# B&R Automation Studio project AS_Target_Simulink_Test (part 2)

### sfc_sdi.h
```c
/* Copyright 2013-2014 The MathWorks, Inc. */

#ifndef _sf_runtime_sf_sdi_h_
#define _sf_runtime_sf_sdi_h_

#ifdef SUPPORTS_PRAGMA_ONCE
#pragma once
#endif

#include "sf_runtime_spec.h"

typedef enum {
    SF_DATA_MODE = 0,
    SF_CHILD_ACTIVITY_MODE  = 0x01,
    SF_LEAF_ACTIVITY_MODE   = 0x02,
    SF_SELF_ACTIVITY_MODE   = 0x04
} SFSdiModeFlag;

typedef enum {
    SF_DATA_TYPE_BEGIN = 0,
    SF_DATA_TYPE_DOUBLE = SF_DATA_TYPE_BEGIN,
    SF_DATA_TYPE_SINGLE,
    SF_DATA_TYPE_INT8,
    SF_DATA_TYPE_UINT8,
    SF_DATA_TYPE_INT16,
    SF_DATA_TYPE_UINT16,
    SF_DATA_TYPE_INT32,
    SF_DATA_TYPE_UINT32,
    SF_DATA_TYPE_BOOLEAN,
    SF_DATA_TYPE_LAST
} SF2SdiBuiltInDataTypes;

typedef enum {
    SF_DIMENSIONS_BEGIN = 0,
    SF_DIMENSIONS_MODE_FIXED = SF_DIMENSIONS_BEGIN,
    SF_DIMENSIONS_MODE_VARIABLE,
    SF_DIMENSIONS_LAST
} SF2SdiDimsMode;

typedef enum {
    SF_COMPLEXITY_BEGIN = 0,
    SF_REAL = SF_COMPLEXITY_BEGIN,
    SF_COMPLEX,
    SF_COMPLEXITY_LAST
} SF2SdiComplexity;

typedef enum {
    SF_SAMPLE_TIME_BEGIN = 0,
    SF_SAMPLE_TIME_CONTINUOUS = SF_SAMPLE_TIME_BEGIN,
    SF_SAMPLE_TIME_DISCRETE,
    SF_SAMPLE_TIME_LAST
} SF2SdiUpdateMethod;

typedef struct SignalExportStruct_t {
    int useCustomName;
    int limitDataPoints;
    int decimate;
    const char* logName;
    const char* signalName;
    unsigned int maxPoints;
    unsigned int decimation;
} SignalExportStruct;

typedef struct sdiBlockID {
    void* SimStruct;
    char* mdlRefFullPath;
    char* blkPath;
    void* sdiRuntime;
} sdiBlockID_t;

LIBMWSF_RUNTIME_API void sdi_database_initialize(struct sdiBlockID* blockId,
                                                 unsigned int* stateSSIDs,
                                                 uint8_T* loggedStatesBuffer, int numStates,
                                                 unsigned int* dataSSIDs,
                                                 uint8_T* loggedDataBuffer, int numData);

LIBMWSF_RUNTIME_API void sdi_database_terminate(struct sdiBlockID* blockId);

LIBMWSF_RUNTIME_API void sdi_register_self_activity_signal(
    struct sdiBlockID* blockId,
    const char* targetName,
    const char* ssid,
    int uMethod,
    SignalExportStruct *sigExportProps,
    unsigned int ssId);

LIBMWSF_RUNTIME_API void sdi_register_child_activity_signal(
    struct sdiBlockID* blockId,
    const char* targetName,
    const char* parentStateRelativePath,
    int numChildStates,
    const char** stateNames,
    int* values,
    int signalSize,
    int uMethod,
    unsigned int ssId);

LIBMWSF_RUNTIME_API void sdi_register_leaf_activity_signal(
    struct sdiBlockID* blockId,
    const char* targetName,
    const char* parentStateRelativePath,
    int numLeafStates,
    const char** stateNames,
    int* values,
    int signalSize,
    int uMethod,
    unsigned int ssId);

LIBMWSF_RUNTIME_API void sdi_register_enum_data_type_signal(
    struct sdiBlockID* blockId,
    const char* targetName,
    const char* parentStateRelativePath,
    const char* enumTypeName,
    int numLiterals,
    const char** literals,
    int* enumValues,
    int storageSize, int isSigned,
    int numDims, int* dimsArray,
    int uMethod,
    int dimsMode,
    int complexity,
    SignalExportStruct *sigExportProps,
    unsigned int ssId);

LIBMWSF_RUNTIME_API void sdi_register_builtin_data_type_signal(
    struct sdiBlockID* blockId,
    const char* targetName,
    const char* parentStateRelativePath,
    int numDims,
    int* dims,
    int updateMethod,
    int typ,
    int dimsMode,
    int complexity,
    SignalExportStruct *sigExportProps,
    const char* units,
    unsigned int ssId);

LIBMWSF_RUNTIME_API void sdi_register_fixed_point_data_type_slope_bias_scaling(
    struct sdiBlockID* blockId,
    const char* targetName,
    const char* parentStateRelativePath,
    int numDims,
    int* dimsArray,
    int uMethod,
    int dimsMode,
    int complexity,
    int numericType,
    unsigned int signedness,
    int wordLength,
    double slopeAdjustFactor,
    int fixedExponent,
    double bias,
    SignalExportStruct *sigExportProps,
    const char* units,
    unsigned int ssId);

LIBMWSF_RUNTIME_API void sdi_register_fixed_point_data_type_binary_point_scaling(
    struct sdiBlockID* blockId,
    const char* targetName,
    const char* parentStateRelativePath,
    int numDims,
    int* dimsArray,
    int uMethod,
    int dimsMode,
    int complexity,
    int numericType,
    unsigned int signedness,
    int wordLength,
    int fractionLength,
    SignalExportStruct *sigExportProps,
    const char* units,
    unsigned int ssId);

LIBMWSF_RUNTIME_API void sdi_register_non_virtual_bus_parent(
    struct sdiBlockID* blockId,
    unsigned int ssId,
    unsigned int busIdx,
    unsigned int parentsIdx,
    unsigned int busSize,
    const char* targetName,
    int numDims,
    int* dimensions);

LIBMWSF_RUNTIME_API void sdi_register_non_virtual_bus_built_in_type_leaf(
    struct sdiBlockID* blockId,
    int uMethod,
    unsigned int ssId,
    unsigned int parentsIdx,
    const char* targetName,
    int numDims,
    int* dimensions,
    int leafComplexity,
    int leafDataType,
    int leafOffset,
    const char* units);

LIBMWSF_RUNTIME_API void sdi_register_non_virtual_bus_fixpt_slope_bias_scaling_type_leaf(
    struct sdiBlockID* blockId,
    int uMethod,
    unsigned int ssId,
    unsigned int parentsIdx,
    const char* targetName,
    int numDims,
    int* dimensions,
    int leafComplexity,
    int numericType,
    unsigned int signedness,
    int wordLength,
    double slopeAdjustFactor,
    int fixedExponent,
    double bias,
    int leafOffset,
    const char* units);

LIBMWSF_RUNTIME_API void sdi_register_non_virtual_bus_fixpt_binary_point_scaling_type_leaf(
    struct sdiBlockID* blockId,
    int uMethod,
    unsigned int ssId,
    unsigned int parentsIdx,
    const char* targetName,
    int numDims,
    int* dimensions,
    int leafComplexity,
    int numericType,
    unsigned int signedness,
    int wordLength,
    int fractionLength,
    int leafOffset,
    const char* units);

LIBMWSF_RUNTIME_API void sdi_register_non_virtual_bus_enum_type_type_leaf(
    struct sdiBlockID* blockId,
    int uMethod,
    unsigned int ssId,
    unsigned int parentsIdx,
    const char* targetName,
    int numDims,
    int* dimensions,
    int leafComplexity,
    const char* enumName,
    int numLiterals,
    const char** literals,
    int* enumValues,
    int storageSize,
    int isSigned,
    int leafOffset);

LIBMWSF_RUNTIME_API void sdi_register_non_virtual_bus(
    struct sdiBlockID* blockId,
    void* busAddr,
    int uMethod,
    const char* targetName,
    const char* parentStateRelativePath,
    int numDims,
    int* dimensions,
    unsigned int busSize,
    SignalExportStruct *sigExportProps,
    unsigned int ssId);

LIBMWSF_RUNTIME_API void sdi_stream_child_activity_signal(struct sdiBlockID* blockId, unsigned int ssId, void* data);
LIBMWSF_RUNTIME_API void sdi_stream_data_signal(struct sdiBlockID* blockId, unsigned int ssId, void* data);
LIBMWSF_RUNTIME_API void sdi_stream_bus_element(struct sdiBlockID* blockId, unsigned int ssId, const char* elementExpr, void* elementData);
LIBMWSF_RUNTIME_API void sdi_update_self_activity_signal(struct sdiBlockID* blockId, unsigned int ssId, int value);
LIBMWSF_RUNTIME_API void sdi_update_leaf_activity_signal(struct sdiBlockID* blockId, unsigned int ssId, int value);
LIBMWSF_RUNTIME_API void sf_rt_strcat_ascii(char* dest, int destMaxLen, char* str1, int maxLen1, char* str2, int maxLen2);

LIBMWSF_RUNTIME_API int cStrcmp(char* arg1, char* arg2);
LIBMWSF_RUNTIME_API int cStrncmp(char* str1, char* str2, int len);
LIBMWSF_RUNTIME_API int cStrlen(char* arg1);

#endif
```

### DebuggerRuntimeInterface.h
```c
/* Copyright 1997-2016 The MathWorks, Inc. */

#ifndef _debugger_codegen_interface_h
#define _debugger_codegen_interface_h

#ifdef SUPPORTS_PRAGMA_ONCE
#pragma once
#endif

#if defined(S_FUNCTION_NAME)
#include "mwmathutil.h"
#endif

#include "sf_runtime/sf_runtime_spec.h"

typedef struct SimStruct_tag SimStruct;

LIBMWSF_RUNTIME_API void* sfListenerInitializeUsingSimStruct(SimStruct* S);
LIBMWSF_RUNTIME_API void* sfListenerInitializeUsingBlockPath(char* blkPath);

LIBMWSF_RUNTIME_API void sfListenerTerminate(void* rt);
LIBMWSF_RUNTIME_API void sfListenerInitializeRuntimeVars(void* rt, int* areListenersActive, int* numFcnVars, char** dataNames[],void** dataPtrs[], char** marshallingOutFcns[], char** marshallingInFcns[],  int* statuses[], int* lineNumber);

LIBMWSF_RUNTIME_API void sfListenerReportScriptName(void* rt, char* aScriptName);

LIBMWSF_RUNTIME_API void sfListenerReportStartingSection(void* rt, unsigned int aSSIDNumber, int aSectionId);
LIBMWSF_RUNTIME_API void sfListenerReportEndingSection(void* rt, unsigned int aSSIDNumber, int aSectionId);

LIBMWSF_RUNTIME_API void sfListenerPushScope(void* rt, unsigned int aSSIDNumber, unsigned int N, char* aVarNames[], void* aDataPtr[], char* aMarchallingOutFunctions[], char* aMarshallingInFunctions[], int aStatus[]);
LIBMWSF_RUNTIME_API void sfListenerPopScope(void* rt, unsigned int aSSIDNumber);

LIBMWSF_RUNTIME_API void sfListenerPushScopeForChart(void* rt, unsigned int aSSIDNumber, unsigned int N, char* aVarNames[], void* aDataPtr[], char* aMarshallingOutFunctions[], char* aMarshallingInFunctions[], int aStatus[]);
LIBMWSF_RUNTIME_API void sfListenerPopScopeForChart(void* rt, unsigned int aSSIDNumber);

LIBMWSF_RUNTIME_API void sfListenerReportStartingEventBroadcast(void* rt, unsigned int aEventSSIDNumber, int aSectionId);
LIBMWSF_RUNTIME_API void sfListenerReportEndingEventBroadcast(void* rt, unsigned int aEventSSIDNumber, int aSectionId);
LIBMWSF_RUNTIME_API void sfListenerReportLineNumber(void* rt, unsigned int aSSIDNumber,int aLineNumber);

LIBMWSF_RUNTIME_API void sfListenerReportScriptName(void* rt, char* scriptName);

#endif
```

### Program Logical/Model/pend_mod (ANSIC, version 1.00.0)

#### global.txt
```
VAR
	    y : ARRAY[0..1] OF LREAL:= [2(0)]; (*Output variables (car position and pendulum angle)*)
	    x : ARRAY[0..3] OF LREAL:= [4(0)]; (*State variables (x, v, theta, omega)*)
	    F : LREAL := 0; (*Manipulated plant input: Force F*)
END_VAR
```

#### pend_mod.c
```c
/********************************************************************
 * COPYRIGHT -- Bernecker + Rainer Industrie-Elektronik Ges.m.b.H.
 ********************************************************************
 * Program: pend_mod_nlin
 * File: pend_mod.c
 * Author: Bernecker + Rainer Industrie Elektronik Ges.m.b.H.
 * Created: Fri Apr 16 22:40:22 2010
 ********************************************************************
 * Implementation of program pend_mod_nlin
 ********************************************************************
 * Generated with B&R Automation Studio Target for Simulink  V6.1.0
 * (ERT based)
 ********************************************************************/

#define _ASMATH_
#define ASMATH_
#define _ASMATH_H
#define ASMATH_H
#define _ASMATH_H_
#define ASMATH_H_
#define _ASSTRING_
#define ASSTRING_
#define _ASSTRING_H
#define ASSTRING_H
#define _ASSTRING_H_
#define ASSTRING_H_
#include <bur/plctypes.h>
#ifdef _DEFAULT_INCLUDES
#include <AsDefault.h>
#endif

#include "pend_mod_nlin.h"
#include "rtwtypes.h"

/*  Defines */

/*  Data Types */

/**************************** GLOBAL DATA *************************************/
/*  Definitions */

/*  Declarations  */

/***************************** FILE SCOPE DATA ********************************/

/*************************** FUNCTIONS ****************************************/
#ifdef __cplusplus

unsigned long bur_heap_size = 6553500;

#endif

  void _INIT mainINIT(void)
{

    UDINT st_ident;
  RTInfo_typ rt_info;
  rt_info.enable = 1;
  RTInfo(&rt_info);
  if (rt_info.cycle_time != 10000) {
    /* cycle time does not match Simulink fixed-step size */
    ST_ident("pend_mod", 0, &st_ident);
    ST_tmp_suspend(st_ident);
    ERR_warning(33310, 0);
  }

  /* initialize model */
  pend_mod_nlin_initialize();

}
void _CYCLIC mainCYCLIC(void)
{
	if(start)
	{/* call model step function */
		pend_mod_nlin_output();
		pend_mod_nlin_update();
	}
	if(reset)
	{
		start = 0;
		pend_mod_nlin_initialize();
		ref = 0;
		x[0] = x[1] = x[2] = x[3] = 0;
		y[0] = y[1] = 0;
		F = 0;
		reset = 0;
	}
}
void _EXIT mainEXIT(void)
{
  /* terminate model */
  pend_mod_nlin_terminate();

} /*****************************************************************************
     Task sample time: 0.01s
   *****************************************************************************/
/*****************************************************************************
   B&R Automation Studio Target for Simulink Version: V6.1.0 (06-Nov-2019)
 *****************************************************************************/

/*======================== TOOL VERSION INFORMATION ==========================*
 * MATLAB 9.7 (R2019b)18-Jul-2019                                             *
 * Simulink 10.0 (R2019b)18-Jul-2019                                          *
 * Simulink Coder 9.2 (R2019b)18-Jul-2019                                     *
 * Embedded Coder 7.3 (R2019b)18-Jul-2019                                     *
 * Stateflow 10.1 (R2019b)18-Jul-2019                                         *
 * Fixed-Point Designer 6.4 (R2019b)18-Jul-2019                               *
 *============================================================================*/

/*======================= LICENSE IN USE INFORMATION =========================*
 * control_toolbox                                                            *
 * matlab                                                                     *
 * matlab_coder                                                               *
 * real-time_workshop                                                         *
 * rtw_embedded_coder                                                         *
 * simulink                                                                   *
 *============================================================================*/
```

#### pend_mod_nlin.c
```c
/********************************************************************
 * COPYRIGHT -- Bernecker + Rainer Industrie-Elektronik Ges.m.b.H.
 ********************************************************************
 * Program: pend_mod_nlin
 * File: pend_mod_nlin.c
 * Author: Bernecker + Rainer Industrie Elektronik Ges.m.b.H.
 * Created: Fri Apr 16 22:40:22 2010
 ********************************************************************
 * Implementation of program pend_mod_nlin
 ********************************************************************
 * Generated with B&R Automation Studio Target for Simulink  V6.1.0
 * (ERT based)
 ********************************************************************/

#include "pend_mod_nlin.h"
#include "pend_mod_nlin_private.h"

/*  Defines */

/*  Data Types */

/**************************** GLOBAL DATA *************************************/
/*  Definitions */

/* Block signals (default storage) */
BlockIO_pend_mod_nlin pend_mod_nlin_B;

/* Continuous states */
ContinuousStates_pend_mod_nlin pend_mod_nlin_X;

/* Real-time model */
RT_MODEL_pend_mod_nlin pend_mod_nlin_M_;
RT_MODEL_pend_mod_nlin *const pend_mod_nlin_M = &pend_mod_nlin_M_;

/*  Declarations  */

/***************************** FILE SCOPE DATA ********************************/

/*************************** FUNCTIONS ****************************************/

/*
 * This function updates continuous states using the ODE1 fixed-step
 * solver algorithm
 */
static void rt_ertODEUpdateContinuousStates(RTWSolverInfo *si )
{
  time_T tnew = rtsiGetSolverStopTime(si);
  time_T h = rtsiGetStepSize(si);
  real_T *x = rtsiGetContStates(si);
  ODE1_IntgData *id = (ODE1_IntgData *)rtsiGetSolverData(si);
  real_T *f0 = id->f[0];
  int_T i;
  int_T nXc = 4;
  rtsiSetSimTimeStep(si,MINOR_TIME_STEP);
  rtsiSetdX(si, f0);
  pend_mod_nlin_derivatives();
  rtsiSetT(si, tnew);
  for (i = 0; i < nXc; ++i) {
    x[i] += h * f0[i];
  }

  rtsiSetSimTimeStep(si,MAJOR_TIME_STEP);
}

/* Model output function */
void pend_mod_nlin_output(void)
{
  real_T x_tmp;
  real_T vdot_tmp;
  real_T vdot_tmp_0;
  if (rtmIsMajorTimeStep(pend_mod_nlin_M)) {
    /* set solver stop time */
    if (!(pend_mod_nlin_M->Timing.clockTick0+1)) {
      rtsiSetSolverStopTime(&pend_mod_nlin_M->solverInfo,
                            ((pend_mod_nlin_M->Timing.clockTickH0 + 1) *
        pend_mod_nlin_M->Timing.stepSize0 * 4294967296.0));
    } else {
      rtsiSetSolverStopTime(&pend_mod_nlin_M->solverInfo,
                            ((pend_mod_nlin_M->Timing.clockTick0 + 1) *
        pend_mod_nlin_M->Timing.stepSize0 + pend_mod_nlin_M->Timing.clockTickH0 *
        pend_mod_nlin_M->Timing.stepSize0 * 4294967296.0));
    }
  }                                    /* end MajorTimeStep */

  /* Update absolute time of base rate at minor time step */
  if (rtmIsMinorTimeStep(pend_mod_nlin_M)) {
    pend_mod_nlin_M->Timing.t[0] = rtsiGetT(&pend_mod_nlin_M->solverInfo);
  }

  /* Integrator: '<S1>/x_dot' */
  pend_mod_nlin_B.x_dot = pend_mod_nlin_X.x_dot_CSTATE;

  /* Integrator: '<S1>/theta_dot' */
  pend_mod_nlin_B.theta_dot = pend_mod_nlin_X.theta_dot_CSTATE;

  /* S-Function (bur_out): '<Root>/Output' */
  y[0] = pend_mod_nlin_B.x_dot;
  y[1] = pend_mod_nlin_B.theta_dot;

  /* Integrator: '<S1>/v_dot' */
  pend_mod_nlin_B.v_dot = pend_mod_nlin_X.v_dot_CSTATE;

  /* Integrator: '<S1>/omega_dot' */
  pend_mod_nlin_B.omega_dot = pend_mod_nlin_X.omega_dot_CSTATE;

  /* S-Function (bur_out): '<Root>/Output1' */
  x[0] = pend_mod_nlin_B.x_dot;
  x[1] = pend_mod_nlin_B.v_dot;
  x[2] = pend_mod_nlin_B.theta_dot;
  x[3] = pend_mod_nlin_B.omega_dot;

  /* S-Function (bur_in): '<Root>/Input' */
  pend_mod_nlin_B.Input = F;

  /* MATLAB Function: '<S1>/Inverted Pendulum  (Non-linear model)' */
  /* MATLAB Function 'inverted_pendulum_embm/Inverted Pendulum  (Non-linear model)': '<S2>:1' */
  /* '<S2>:1:4' */
  x_tmp = sin(pend_mod_nlin_B.theta_dot);
  vdot_tmp = cos(pend_mod_nlin_B.theta_dot);
  vdot_tmp_0 = x_tmp * x_tmp * 0.1 + 1000.0;
  pend_mod_nlin_B.vdot = ((pend_mod_nlin_B.omega_dot * pend_mod_nlin_B.omega_dot
    * 0.05 * x_tmp + -0.98100000000000009 * x_tmp * vdot_tmp) +
    pend_mod_nlin_B.Input) / vdot_tmp_0;

  /* '<S2>:1:5' */
  pend_mod_nlin_B.omegadot = (((9810.9810000000016 * x_tmp - 0.0 *
    pend_mod_nlin_B.omega_dot) - vdot_tmp * pend_mod_nlin_B.Input) -
    pend_mod_nlin_B.omega_dot * pend_mod_nlin_B.omega_dot * 0.05 * sin
    (pend_mod_nlin_B.theta_dot) * vdot_tmp) / vdot_tmp_0 / 0.5;
  if (rtmIsMajorTimeStep(pend_mod_nlin_M)) {
  }
}

/* Model update function */
void pend_mod_nlin_update(void)
{
  if (rtmIsMajorTimeStep(pend_mod_nlin_M)) {
    rt_ertODEUpdateContinuousStates(&pend_mod_nlin_M->solverInfo);
  }

  /* Update absolute time for base rate */
  /* The "clockTick0" counts the number of times the code of this task has
   * been executed. The absolute time is the multiplication of "clockTick0"
   * and "Timing.stepSize0". Size of "clockTick0" ensures timer will not
   * overflow during the application lifespan selected.
   * Timer of this task consists of two 32 bit unsigned integers.
   * The two integers represent the low bits Timing.clockTick0 and the high bits
   * Timing.clockTickH0. When the low bit overflows to 0, the high bits increment.
   */
  if (!(++pend_mod_nlin_M->Timing.clockTick0)) {
    ++pend_mod_nlin_M->Timing.clockTickH0;
  }

  pend_mod_nlin_M->Timing.t[0] = rtsiGetSolverStopTime
    (&pend_mod_nlin_M->solverInfo);

  {
    /* Update absolute timer for sample time: [0.01s, 0.0s] */
    /* The "clockTick1" counts the number of times the code of this task has
     * been executed. The resolution of this integer timer is 0.01, which is the step size
     * of the task. Size of "clockTick1" ensures timer will not overflow during the
     * application lifespan selected.
     * Timer of this task consists of two 32 bit unsigned integers.
     * The two integers represent the low bits Timing.clockTick1 and the high bits
     * Timing.clockTickH1. When the low bit overflows to 0, the high bits increment.
     */
    pend_mod_nlin_M->Timing.clockTick1++;
    if (!pend_mod_nlin_M->Timing.clockTick1) {
      pend_mod_nlin_M->Timing.clockTickH1++;
    }
  }
}

/* Derivatives for root system: '<Root>' */
void pend_mod_nlin_derivatives(void)
{
  StateDerivatives_pend_mod_nlin *_rtXdot;
  _rtXdot = ((StateDerivatives_pend_mod_nlin *) pend_mod_nlin_M->derivs);

  /* Derivatives for Integrator: '<S1>/x_dot' */
  _rtXdot->x_dot_CSTATE = pend_mod_nlin_B.v_dot;

  /* Derivatives for Integrator: '<S1>/theta_dot' */
  _rtXdot->theta_dot_CSTATE = pend_mod_nlin_B.omega_dot;

  /* Derivatives for Integrator: '<S1>/v_dot' */
  _rtXdot->v_dot_CSTATE = pend_mod_nlin_B.vdot;

  /* Derivatives for Integrator: '<S1>/omega_dot' */
  _rtXdot->omega_dot_CSTATE = pend_mod_nlin_B.omegadot;
}

/* Model initialize function */
void pend_mod_nlin_initialize(void)
{
  /* Registration code */
  {
    /* Setup solver object */
    rtsiSetSimTimeStepPtr(&pend_mod_nlin_M->solverInfo,
                          &pend_mod_nlin_M->Timing.simTimeStep);
    rtsiSetTPtr(&pend_mod_nlin_M->solverInfo, &rtmGetTPtr(pend_mod_nlin_M));
    rtsiSetStepSizePtr(&pend_mod_nlin_M->solverInfo,
                       &pend_mod_nlin_M->Timing.stepSize0);
    rtsiSetdXPtr(&pend_mod_nlin_M->solverInfo, &pend_mod_nlin_M->derivs);
    rtsiSetContStatesPtr(&pend_mod_nlin_M->solverInfo, (real_T **)
                         &pend_mod_nlin_M->contStates);
    rtsiSetNumContStatesPtr(&pend_mod_nlin_M->solverInfo,
      &pend_mod_nlin_M->Sizes.numContStates);
    rtsiSetNumPeriodicContStatesPtr(&pend_mod_nlin_M->solverInfo,
      &pend_mod_nlin_M->Sizes.numPeriodicContStates);
    rtsiSetPeriodicContStateIndicesPtr(&pend_mod_nlin_M->solverInfo,
      &pend_mod_nlin_M->periodicContStateIndices);
    rtsiSetPeriodicContStateRangesPtr(&pend_mod_nlin_M->solverInfo,
      &pend_mod_nlin_M->periodicContStateRanges);
    rtsiSetErrorStatusPtr(&pend_mod_nlin_M->solverInfo, (&rtmGetErrorStatus
      (pend_mod_nlin_M)));
    rtsiSetRTModelPtr(&pend_mod_nlin_M->solverInfo, pend_mod_nlin_M);
  }

  rtsiSetSimTimeStep(&pend_mod_nlin_M->solverInfo, MAJOR_TIME_STEP);
  pend_mod_nlin_M->intgData.f[0] = pend_mod_nlin_M->odeF[0];
  pend_mod_nlin_M->contStates = ((ContinuousStates_pend_mod_nlin *)
    &pend_mod_nlin_X);
  rtsiSetSolverData(&pend_mod_nlin_M->solverInfo, (void *)
                    &pend_mod_nlin_M->intgData);
  rtsiSetSolverName(&pend_mod_nlin_M->solverInfo,"ode1");
  rtmSetTPtr(pend_mod_nlin_M, &pend_mod_nlin_M->Timing.tArray[0]);
  pend_mod_nlin_M->Timing.stepSize0 = 0.01;

  /* InitializeConditions for Integrator: '<S1>/x_dot' */
  pend_mod_nlin_X.x_dot_CSTATE = 0.0;

  /* InitializeConditions for Integrator: '<S1>/theta_dot' */
  pend_mod_nlin_X.theta_dot_CSTATE = 0.01;

  /* InitializeConditions for Integrator: '<S1>/v_dot' */
  pend_mod_nlin_X.v_dot_CSTATE = 0.0;

  /* InitializeConditions for Integrator: '<S1>/omega_dot' */
  pend_mod_nlin_X.omega_dot_CSTATE = 0.0;
}

/* Model terminate function */
void pend_mod_nlin_terminate(void)
{
  /* (no terminate code required) */
}

/*======================== TOOL VERSION INFORMATION ==========================*
 * MATLAB 9.7 (R2019b)18-Jul-2019                                             *
 * Simulink 10.0 (R2019b)18-Jul-2019                                          *
 * Simulink Coder 9.2 (R2019b)18-Jul-2019                                     *
 * Embedded Coder 7.3 (R2019b)18-Jul-2019                                     *
 * Stateflow 10.1 (R2019b)18-Jul-2019                                         *
 * Fixed-Point Designer 6.4 (R2019b)18-Jul-2019                               *
 *============================================================================*/

/*======================= LICENSE IN USE INFORMATION =========================*
 * control_toolbox                                                            *
 * matlab                                                                     *
 * matlab_coder                                                               *
 * real-time_workshop                                                         *
 * rtw_embedded_coder                                                         *
 * simulink                                                                   *
 *============================================================================*/
```

#### pend_mod_nlin.h
```c
/********************************************************************
 * COPYRIGHT -- Bernecker + Rainer Industrie-Elektronik Ges.m.b.H.
 ********************************************************************
 * Program: pend_mod_nlin
 * File: pend_mod_nlin.h
 * Author: Bernecker + Rainer Industrie Elektronik Ges.m.b.H.
 * Created: Fri Apr 16 22:40:22 2010
 ********************************************************************
 * Header for program pend_mod_nlin
 ********************************************************************
 * Generated with B&R Automation Studio Target for Simulink  V6.1.0
 * (ERT based)
 ********************************************************************/

#ifndef RTW_HEADER_pend_mod_nlin_h_
#define RTW_HEADER_pend_mod_nlin_h_
#include <math.h>
#ifndef pend_mod_nlin_COMMON_INCLUDES_
# define pend_mod_nlin_COMMON_INCLUDES_
#include "rtwtypes.h"
#include "rtw_continuous.h"
#include "rtw_solver.h"
#endif                                 /* pend_mod_nlin_COMMON_INCLUDES_ */

#include <bur/plctypes.h>

#ifdef _DEFAULT_INCLUDES
 #include <AsDefault.h>
#endif

#ifndef AST_ROUND
#define AST_ROUND(x) ((x)>=0?(long long)((x)+0.5):(long long)((x)-0.5))
#endif

#include "pend_mod_nlin_types.h"

/* Macros for accessing real-time model data structure */
#ifndef rtmGetContStateDisabled
# define rtmGetContStateDisabled(rtm)  ((rtm)->contStateDisabled)
#endif

#ifndef rtmSetContStateDisabled
# define rtmSetContStateDisabled(rtm, val) ((rtm)->contStateDisabled = (val))
#endif

#ifndef rtmGetContStates
# define rtmGetContStates(rtm)         ((rtm)->contStates)
#endif

#ifndef rtmSetContStates
# define rtmSetContStates(rtm, val)    ((rtm)->contStates = (val))
#endif

#ifndef rtmGetContTimeOutputInconsistentWithStateAtMajorStepFlag
# define rtmGetContTimeOutputInconsistentWithStateAtMajorStepFlag(rtm) ((rtm)->CTOutputIncnstWithState)
#endif

#ifndef rtmSetContTimeOutputInconsistentWithStateAtMajorStepFlag
# define rtmSetContTimeOutputInconsistentWithStateAtMajorStepFlag(rtm, val) ((rtm)->CTOutputIncnstWithState = (val))
#endif

#ifndef rtmGetDerivCacheNeedsReset
# define rtmGetDerivCacheNeedsReset(rtm) ((rtm)->derivCacheNeedsReset)
#endif

#ifndef rtmSetDerivCacheNeedsReset
# define rtmSetDerivCacheNeedsReset(rtm, val) ((rtm)->derivCacheNeedsReset = (val))
#endif

#ifndef rtmGetIntgData
# define rtmGetIntgData(rtm)           ((rtm)->intgData)
#endif

#ifndef rtmSetIntgData
# define rtmSetIntgData(rtm, val)      ((rtm)->intgData = (val))
#endif

#ifndef rtmGetOdeF
# define rtmGetOdeF(rtm)               ((rtm)->odeF)
#endif

#ifndef rtmSetOdeF
# define rtmSetOdeF(rtm, val)          ((rtm)->odeF = (val))
#endif

#ifndef rtmGetPeriodicContStateIndices
# define rtmGetPeriodicContStateIndices(rtm) ((rtm)->periodicContStateIndices)
#endif

#ifndef rtmSetPeriodicContStateIndices
# define rtmSetPeriodicContStateIndices(rtm, val) ((rtm)->periodicContStateIndices = (val))
#endif

#ifndef rtmGetPeriodicContStateRanges
# define rtmGetPeriodicContStateRanges(rtm) ((rtm)->periodicContStateRanges)
#endif

#ifndef rtmSetPeriodicContStateRanges
# define rtmSetPeriodicContStateRanges(rtm, val) ((rtm)->periodicContStateRanges = (val))
#endif

#ifndef rtmGetZCCacheNeedsReset
# define rtmGetZCCacheNeedsReset(rtm)  ((rtm)->zCCacheNeedsReset)
#endif

#ifndef rtmSetZCCacheNeedsReset
# define rtmSetZCCacheNeedsReset(rtm, val) ((rtm)->zCCacheNeedsReset = (val))
#endif

#ifndef rtmGetdX
# define rtmGetdX(rtm)                 ((rtm)->derivs)
#endif

#ifndef rtmSetdX
# define rtmSetdX(rtm, val)            ((rtm)->derivs = (val))
#endif

#ifndef rtmGetErrorStatus
# define rtmGetErrorStatus(rtm)        ((rtm)->errorStatus)
#endif

#ifndef rtmSetErrorStatus
# define rtmSetErrorStatus(rtm, val)   ((rtm)->errorStatus = (val))
#endif

#ifndef rtmGetStopRequested
# define rtmGetStopRequested(rtm)      ((rtm)->Timing.stopRequestedFlag)
#endif

#ifndef rtmSetStopRequested
# define rtmSetStopRequested(rtm, val) ((rtm)->Timing.stopRequestedFlag = (val))
#endif

#ifndef rtmGetStopRequestedPtr
# define rtmGetStopRequestedPtr(rtm)   (&((rtm)->Timing.stopRequestedFlag))
#endif

#ifndef rtmGetT
# define rtmGetT(rtm)                  (rtmGetTPtr((rtm))[0])
#endif

#ifndef rtmGetTPtr
# define rtmGetTPtr(rtm)               ((rtm)->Timing.t)
#endif

#ifndef MIN
#define MIN(a,b)                       ((a) < (b) ? (a) : (b))
#endif

#ifndef MAX
#define MAX(a,b)                       ((a) > (b) ? (a) : (b))
#endif

/* Block signals (default storage) */
typedef struct {
  real_T x_dot;                        /* '<S1>/x_dot' */
  real_T theta_dot;                    /* '<S1>/theta_dot' */
  real_T v_dot;                        /* '<S1>/v_dot' */
  real_T omega_dot;                    /* '<S1>/omega_dot' */
  real_T Input;                        /* '<Root>/Input' */
  real_T vdot;                /* '<S1>/Inverted Pendulum  (Non-linear model)' */
  real_T omegadot;            /* '<S1>/Inverted Pendulum  (Non-linear model)' */
} BlockIO_pend_mod_nlin;

/* Continuous states (default storage) */
typedef struct {
  real_T x_dot_CSTATE;                 /* '<S1>/x_dot' */
  real_T theta_dot_CSTATE;             /* '<S1>/theta_dot' */
  real_T v_dot_CSTATE;                 /* '<S1>/v_dot' */
  real_T omega_dot_CSTATE;             /* '<S1>/omega_dot' */
} ContinuousStates_pend_mod_nlin;

/* State derivatives (default storage) */
typedef struct {
  real_T x_dot_CSTATE;                 /* '<S1>/x_dot' */
  real_T theta_dot_CSTATE;             /* '<S1>/theta_dot' */
  real_T v_dot_CSTATE;                 /* '<S1>/v_dot' */
  real_T omega_dot_CSTATE;             /* '<S1>/omega_dot' */
} StateDerivatives_pend_mod_nlin;

/* State disabled  */
typedef struct {
  boolean_T x_dot_CSTATE;              /* '<S1>/x_dot' */
  boolean_T theta_dot_CSTATE;          /* '<S1>/theta_dot' */
  boolean_T v_dot_CSTATE;              /* '<S1>/v_dot' */
  boolean_T omega_dot_CSTATE;          /* '<S1>/omega_dot' */
} StateDisabled_pend_mod_nlin;

#ifndef ODE1_INTG
#define ODE1_INTG

/* ODE1 Integration Data */
typedef struct {
  real_T *f[1];                        /* derivatives */
} ODE1_IntgData;

#endif

/* Real-time Model Data Structure */
struct tag_RTM_pend_mod_nlin {
  const char_T *errorStatus;
  RTWSolverInfo solverInfo;
  ContinuousStates_pend_mod_nlin *contStates;
  int_T *periodicContStateIndices;
  real_T *periodicContStateRanges;
  real_T *derivs;
  boolean_T *contStateDisabled;
  boolean_T zCCacheNeedsReset;
  boolean_T derivCacheNeedsReset;
  boolean_T CTOutputIncnstWithState;
  real_T odeF[1][4];
  ODE1_IntgData intgData;

  /*
   * Sizes:
   * The following substructure contains sizes information
   * for many of the model attributes such as inputs, outputs,
   * dwork, sample times, etc.
   */
  struct {
    int_T numContStates;
    int_T numPeriodicContStates;
    int_T numSampTimes;
  } Sizes;

  /*
   * Timing:
   * The following substructure contains information regarding
   * the timing information for the model.
   */
  struct {
    uint32_T clockTick0;
    uint32_T clockTickH0;
    time_T stepSize0;
    uint32_T clockTick1;
    uint32_T clockTickH1;
    SimTimeStep simTimeStep;
    boolean_T stopRequestedFlag;
    time_T *t;
    time_T tArray[2];
  } Timing;
};

/* Block signals (default storage) */
extern BlockIO_pend_mod_nlin pend_mod_nlin_B;

/* Continuous states (default storage) */
extern ContinuousStates_pend_mod_nlin pend_mod_nlin_X;

/* Model entry point functions */
extern void pend_mod_nlin_initialize(void);
extern void pend_mod_nlin_output(void);
extern void pend_mod_nlin_update(void);
extern void pend_mod_nlin_terminate(void);

/* Real-time Model object */
extern RT_MODEL_pend_mod_nlin *const pend_mod_nlin_M;

/*-
 * The generated code includes comments that allow you to trace directly
 * back to the appropriate location in the model.  The basic format
 * is <system>/block_name, where system is the system number (uniquely
 * assigned by Simulink) and block_name is the name of the block.
 *
 * Use the MATLAB hilite_system command to trace the generated code back
 * to the model.  For example,
 *
 * hilite_system('<S3>')    - opens system 3
 * hilite_system('<S3>/Kp') - opens and selects block Kp which resides in S3
 *
 * Here is the system hierarchy for this model
 *
 * '<Root>' : 'pend_mod_nlin'
 * '<S1>'   : 'pend_mod_nlin/inverted_pendulum_embm'
 * '<S2>'   : 'pend_mod_nlin/inverted_pendulum_embm/Inverted Pendulum  (Non-linear model)'
 */
#endif                                 /* RTW_HEADER_pend_mod_nlin_h_ */
```

#### pend_mod_nlin_private.h
```c
/********************************************************************
 * COPYRIGHT -- Bernecker + Rainer Industrie-Elektronik Ges.m.b.H.
 ********************************************************************
 * Program: pend_mod_nlin
 * File: pend_mod_nlin_private.h
 * Author: Bernecker + Rainer Industrie Elektronik Ges.m.b.H.
 * Created: Fri Apr 16 22:40:22 2010
 ********************************************************************
 * Header for program pend_mod_nlin
 ********************************************************************
 * Generated with B&R Automation Studio Target for Simulink  V6.1.0
 * (ERT based)
 ********************************************************************/

#ifndef RTW_HEADER_pend_mod_nlin_private_h_
#define RTW_HEADER_pend_mod_nlin_private_h_
#include "rtwtypes.h"
#define _ASMATH_
#define ASMATH_
#define _ASMATH_H
#define ASMATH_H
#define _ASMATH_H_
#define ASMATH_H_
#define _ASSTRING_
#define ASSTRING_
#define _ASSTRING_H
#define ASSTRING_H
#define _ASSTRING_H_
#define ASSTRING_H_
#include <bur/plctypes.h>
#ifdef _DEFAULT_INCLUDES
#include <AsDefault.h>
#endif

/* Private macros used by the generated code to access rtModel */
#ifndef rtmIsMajorTimeStep
# define rtmIsMajorTimeStep(rtm)       (((rtm)->Timing.simTimeStep) == MAJOR_TIME_STEP)
#endif

#ifndef rtmIsMinorTimeStep
# define rtmIsMinorTimeStep(rtm)       (((rtm)->Timing.simTimeStep) == MINOR_TIME_STEP)
#endif

#ifndef rtmSetTPtr
# define rtmSetTPtr(rtm, val)          ((rtm)->Timing.t = (val))
#endif

#ifndef MIN
#define MIN(a,b)                       ((a) < (b) ? (a) : (b))
#endif

#ifndef MAX
#define MAX(a,b)                       ((a) > (b) ? (a) : (b))
#endif

/* private model entry point functions */
extern void pend_mod_nlin_derivatives(void);

#endif                                 /* RTW_HEADER_pend_mod_nlin_private_h_ */
```

#### pend_mod_nlin_types.h
```c
/********************************************************************
 * COPYRIGHT -- Bernecker + Rainer Industrie-Elektronik Ges.m.b.H.
 ********************************************************************
 * Program: pend_mod_nlin
 * File: pend_mod_nlin_types.h
 * Author: Bernecker + Rainer Industrie Elektronik Ges.m.b.H.
 * Created: Fri Apr 16 22:40:22 2010
 ********************************************************************
 * Header for program pend_mod_nlin
 ********************************************************************
 * Generated with B&R Automation Studio Target for Simulink  V6.1.0
 * (ERT based)
 ********************************************************************/

#ifndef RTW_HEADER_pend_mod_nlin_types_h_
#define RTW_HEADER_pend_mod_nlin_types_h_
#ifndef MIN
#define MIN(a,b)                       ((a) < (b) ? (a) : (b))
#endif

#ifndef MAX
#define MAX(a,b)                       ((a) > (b) ? (a) : (b))
#endif

/* Forward declaration for rtModel */
typedef struct tag_RTM_pend_mod_nlin RT_MODEL_pend_mod_nlin;

#endif                                 /* RTW_HEADER_pend_mod_nlin_types_h_ */
```

#### rtwtypes.h
```c
/********************************************************************
 * COPYRIGHT -- Bernecker + Rainer Industrie-Elektronik Ges.m.b.H.
 ********************************************************************
 * Program: pend_mod_nlin
 * File: rtwtypes.h
 * Author: Bernecker + Rainer Industrie Elektronik Ges.m.b.H.
 * Created: Fri Apr 16 22:40:22 2010
 ********************************************************************
 * Header for program pend_mod_nlin
 ********************************************************************
 * Generated with B&R Automation Studio Target for Simulink  V6.1.0
 * (ERT based)
 ********************************************************************/

#ifndef RTWTYPES_H
#define RTWTYPES_H

/* Logical type definitions */
#if (!defined(__cplusplus))
#  ifndef false
#   define false                       (0U)
#  endif

#  ifndef true
#   define true                        (1U)
#  endif
#endif

/*=======================================================================*
 * Target hardware information
 *   Device type: Intel->x86/Pentium
 *   Number of bits:     char:   8    short:   16    long:  32
 *                       long:  32
 *                       native word size:  32
 *   Byte ordering: LittleEndian
 *   Signed integer division rounds to: Zero
 *   Shift right on a signed integer as arithmetic shift: on
 *=======================================================================*/

/*=======================================================================*
 * Fixed width word size data types:                                     *
 *   int8_T, int16_T, int32_T     - signed 8, 16, or 32 bit integers     *
 *   uint8_T, uint16_T, uint32_T  - unsigned 8, 16, or 32 bit integers   *
 *   real32_T, real64_T           - 32 and 64 bit floating point numbers *
 *=======================================================================*/
typedef signed char int8_T;
typedef unsigned char uint8_T;
typedef short int16_T;
typedef unsigned short uint16_T;
typedef long int32_T;
typedef unsigned long uint32_T;
typedef float real32_T;
typedef double real64_T;

/*===========================================================================*
 * Generic type definitions: boolean_T, char_T, byte_T, int_T, uint_T,       *
 *                           real_T, time_T, ulong_T.                        *
 *===========================================================================*/
typedef double real_T;
typedef double time_T;
typedef unsigned char boolean_T;
typedef long int_T;
typedef unsigned long uint_T;
typedef unsigned long ulong_T;
typedef char char_T;
typedef unsigned char uchar_T;
typedef char_T byte_T;

/*=======================================================================*
 * Min and Max:                                                          *
 *   int8_T, int16_T, int32_T     - signed 8, 16, or 32 bit integers     *
 *   uint8_T, uint16_T, uint32_T  - unsigned 8, 16, or 32 bit integers   *
 *=======================================================================*/
#define MAX_int8_T                     ((int8_T)(127))
#define MIN_int8_T                     ((int8_T)(-128))
#define MAX_uint8_T                    ((uint8_T)(255U))
#define MAX_int16_T                    ((int16_T)(32767))
#define MIN_int16_T                    ((int16_T)(-32768))
#define MAX_uint16_T                   ((uint16_T)(65535U))
#define MAX_int32_T                    ((int32_T)(2147483647))
#define MIN_int32_T                    ((int32_T)(-2147483647-1))
#define MAX_uint32_T                   ((uint32_T)(0xFFFFFFFFU))

/* Block D-Work pointer type */
typedef void * pointer_T;

#endif                                 /* RTWTYPES_H */

#ifndef MIN
#define MIN(a,b)                       ((a) < (b) ? (a) : (b))
#endif

#ifndef MAX
#define MAX(a,b)                       ((a) > (b) ? (a) : (b))
#endif
```

#### task_properties.txt
```
For manual assignment to hardware configuration please
add the following additional include directories:

\Logical\MATLAB_includes\R2019b\

And the following additional build options:

-lm -D MODEL=pend_mod_nlin -D NUMST=2 -D NCSTATES=4 -D HAVESTDIO -D MODEL_HAS_DYNAMICALLY_LOADED_SFCNS=0 -D CLASSIC_INTERFACE=0 -D ALLOCATIONFCN=0 -D TID01EQ=1 -D TERMFCN=1 -D ONESTEPFCN=0 -D MAT_FILE=0 -D MULTI_INSTANCE_CODE=0 -D INTEGER_CODE=0 -D MT=0
```

### Program Logical/Controller/pend_ctrl (ANSIC, version 1.00.0)

#### local.var
```iecst
VAR
	signal : BOOL;
END_VAR
```

#### pend_ctrl.c
```c
/********************************************************************
 * COPYRIGHT -- Bernecker + Rainer Industrie-Elektronik Ges.m.b.H.
 ********************************************************************
 * Program: pend_ctrl_lin
 * File: pend_ctrl.c
 * Author: Bernecker + Rainer Industrie Elektronik Ges.m.b.H.
 * Created: Wed Mar 17 14:21:47 2010
 ********************************************************************
 * Implementation of program pend_ctrl_lin
 ********************************************************************
 * Generated with B&R Automation Studio Target for Simulink  V6.1.0
 * (ERT based)
 ********************************************************************/

#define _ASMATH_
#define ASMATH_
#define _ASMATH_H
#define ASMATH_H
#define _ASMATH_H_
#define ASMATH_H_
#define _ASSTRING_
#define ASSTRING_
#define _ASSTRING_H
#define ASSTRING_H
#define _ASSTRING_H_
#define ASSTRING_H_
#include <bur/plctypes.h>
#ifdef _DEFAULT_INCLUDES
#include <AsDefault.h>
#endif

#include "pend_ctrl_lin.h"
#include "rtwtypes.h"

/*  Defines */

/*  Data Types */

/**************************** GLOBAL DATA *************************************/
/*  Definitions */

/*  Declarations  */

/***************************** FILE SCOPE DATA ********************************/

/*************************** FUNCTIONS ****************************************/
#ifdef __cplusplus

unsigned long bur_heap_size = 6553500;

#endif

  void _INIT mainINIT(void)
{

    UDINT st_ident;
  RTInfo_typ rt_info;
  rt_info.enable = 1;
  RTInfo(&rt_info);
  if (rt_info.cycle_time != 10000) {
    /* cycle time does not match Simulink fixed-step size */
    ST_ident("pend_ctrl", 0, &st_ident);
    ST_tmp_suspend(st_ident);
    ERR_warning(33310, 0);
  }

  /* initialize model */
  pend_ctrl_lin_initialize();

}
void _CYCLIC mainCYCLIC(void)
{
	if(start)
	{
		/* call model step function */
		pend_ctrl_lin_output();
		pend_ctrl_lin_update();
	}

}
void _EXIT mainEXIT(void)
{
  /* terminate model */
  pend_ctrl_lin_terminate();

} /*****************************************************************************
     Task sample time: 0.01s
   *****************************************************************************/
/*****************************************************************************
   B&R Automation Studio Target for Simulink Version: V6.1.0 (06-Nov-2019)
 *****************************************************************************/

/*======================== TOOL VERSION INFORMATION ==========================*
 * MATLAB 9.7 (R2019b)18-Jul-2019                                             *
 * Simulink 10.0 (R2019b)18-Jul-2019                                          *
 * Simulink Coder 9.2 (R2019b)18-Jul-2019                                     *
 * Embedded Coder 7.3 (R2019b)18-Jul-2019                                     *
 * Stateflow 10.1 (R2019b)18-Jul-2019                                         *
 * Fixed-Point Designer 6.4 (R2019b)18-Jul-2019                               *
 *============================================================================*/

/*======================= LICENSE IN USE INFORMATION =========================*
 * control_toolbox                                                            *
 * matlab                                                                     *
 * matlab_coder                                                               *
 * real-time_workshop                                                         *
 * rtw_embedded_coder                                                         *
 * simulink                                                                   *
 *============================================================================*/
```

#### pend_ctrl_lin.c
```c
/********************************************************************
 * COPYRIGHT -- Bernecker + Rainer Industrie-Elektronik Ges.m.b.H.
 ********************************************************************
 * Program: pend_ctrl_lin
 * File: pend_ctrl_lin.c
 * Author: Bernecker + Rainer Industrie Elektronik Ges.m.b.H.
 * Created: Wed Mar 17 14:21:47 2010
 ********************************************************************
 * Implementation of program pend_ctrl_lin
 ********************************************************************
 * Generated with B&R Automation Studio Target for Simulink  V6.1.0
 * (ERT based)
 ********************************************************************/

#include "pend_ctrl_lin.h"
#include "pend_ctrl_lin_private.h"

/*  Defines */

/*  Data Types */

/**************************** GLOBAL DATA *************************************/
/*  Definitions */

/* Block signals (default storage) */
BlockIO_pend_ctrl_lin pend_ctrl_lin_B;

/* Real-time model */
RT_MODEL_pend_ctrl_lin pend_ctrl_lin_M_;
RT_MODEL_pend_ctrl_lin *const pend_ctrl_lin_M = &pend_ctrl_lin_M_;

/*  Declarations  */

/***************************** FILE SCOPE DATA ********************************/

/*************************** FUNCTIONS ****************************************/

/* Model output function */
void pend_ctrl_lin_output(void)
{
  real_T tmp;

  /* S-Function (bur_in): '<S1>/Input' */
  pend_ctrl_lin_B.Input = ref;

  /* Gain: '<S4>/Feed-Forward' */
  pend_ctrl_lin_B.FeedForward = -2987.4616903679112 * pend_ctrl_lin_B.Input;

  /* S-Function (bur_in): '<S3>/Input' */
  pend_ctrl_lin_B.Input_f[0] = x[0];
  pend_ctrl_lin_B.Input_f[1] = x[1];
  pend_ctrl_lin_B.Input_f[2] = x[2];
  pend_ctrl_lin_B.Input_f[3] = x[3];

  /* Gain: '<S4>/LQR Controller' */
  tmp = -2987.4616903679125 * pend_ctrl_lin_B.Input_f[0];
  tmp += -3740.1178916812455 * pend_ctrl_lin_B.Input_f[1];
  tmp += -32774.860875805127 * pend_ctrl_lin_B.Input_f[2];
  tmp += -7399.4348019785593 * pend_ctrl_lin_B.Input_f[3];
  pend_ctrl_lin_B.LQRController = tmp;

  /* Sum: '<S4>/Sum' */
  pend_ctrl_lin_B.Sum = pend_ctrl_lin_B.FeedForward -
    pend_ctrl_lin_B.LQRController;

  /* S-Function (bur_in): '<S3>/Input1' */
  pend_ctrl_lin_B.Input1[0] = y[0];
  pend_ctrl_lin_B.Input1[1] = y[1];

  /* S-Function (bur_out): '<S3>/Output' */
  F = pend_ctrl_lin_B.Sum;
}

/* Model update function */
void pend_ctrl_lin_update(void)
{
  /* (no update code required) */
}

/* Model initialize function */
void pend_ctrl_lin_initialize(void)
{
  /* (no initialization code required) */
}

/* Model terminate function */
void pend_ctrl_lin_terminate(void)
{
  /* (no terminate code required) */
}

/*======================== TOOL VERSION INFORMATION ==========================*
 * MATLAB 9.7 (R2019b)18-Jul-2019                                             *
 * Simulink 10.0 (R2019b)18-Jul-2019                                          *
 * Simulink Coder 9.2 (R2019b)18-Jul-2019                                     *
 * Embedded Coder 7.3 (R2019b)18-Jul-2019                                     *
 * Stateflow 10.1 (R2019b)18-Jul-2019                                         *
 * Fixed-Point Designer 6.4 (R2019b)18-Jul-2019                               *
 *============================================================================*/

/*======================= LICENSE IN USE INFORMATION =========================*
 * control_toolbox                                                            *
 * matlab                                                                     *
 * matlab_coder                                                               *
 * real-time_workshop                                                         *
 * rtw_embedded_coder                                                         *
 * simulink                                                                   *
 *============================================================================*/
```

#### pend_ctrl_lin.h
```c
/********************************************************************
 * COPYRIGHT -- Bernecker + Rainer Industrie-Elektronik Ges.m.b.H.
 ********************************************************************
 * Program: pend_ctrl_lin
 * File: pend_ctrl_lin.h
 * Author: Bernecker + Rainer Industrie Elektronik Ges.m.b.H.
 * Created: Wed Mar 17 14:21:47 2010
 ********************************************************************
 * Header for program pend_ctrl_lin
 ********************************************************************
 * Generated with B&R Automation Studio Target for Simulink  V6.1.0
 * (ERT based)
 ********************************************************************/

#ifndef RTW_HEADER_pend_ctrl_lin_h_
#define RTW_HEADER_pend_ctrl_lin_h_
#ifndef pend_ctrl_lin_COMMON_INCLUDES_
# define pend_ctrl_lin_COMMON_INCLUDES_
#include "rtwtypes.h"
#include "rtw_continuous.h"
#include "rtw_solver.h"
#endif                                 /* pend_ctrl_lin_COMMON_INCLUDES_ */

#include <bur/plctypes.h>

#ifdef _DEFAULT_INCLUDES
 #include <AsDefault.h>
#endif

#ifndef AST_ROUND
#define AST_ROUND(x) ((x)>=0?(long long)((x)+0.5):(long long)((x)-0.5))
#endif

#include "pend_ctrl_lin_types.h"

/* Macros for accessing real-time model data structure */
#ifndef rtmGetErrorStatus
# define rtmGetErrorStatus(rtm)        ((rtm)->errorStatus)
#endif

#ifndef rtmSetErrorStatus
# define rtmSetErrorStatus(rtm, val)   ((rtm)->errorStatus = (val))
#endif

#ifndef MIN
#define MIN(a,b)                       ((a) < (b) ? (a) : (b))
#endif

#ifndef MAX
#define MAX(a,b)                       ((a) > (b) ? (a) : (b))
#endif

/* Block signals (default storage) */
typedef struct {
  real_T Input;                        /* '<S1>/Input' */
  real_T FeedForward;                  /* '<S4>/Feed-Forward' */
  real_T Input_f[4];                   /* '<S3>/Input' */
  real_T LQRController;                /* '<S4>/LQR Controller' */
  real_T Sum;                          /* '<S4>/Sum' */
  real_T Input1[2];                    /* '<S3>/Input1' */
} BlockIO_pend_ctrl_lin;

/* Real-time Model Data Structure */
struct tag_RTM_pend_ctrl_lin {
  const char_T *errorStatus;
};

/* Block signals (default storage) */
extern BlockIO_pend_ctrl_lin pend_ctrl_lin_B;

/* Model entry point functions */
extern void pend_ctrl_lin_initialize(void);
extern void pend_ctrl_lin_output(void);
extern void pend_ctrl_lin_update(void);
extern void pend_ctrl_lin_terminate(void);

/* Real-time Model object */
extern RT_MODEL_pend_ctrl_lin *const pend_ctrl_lin_M;

/*-
 * The generated code includes comments that allow you to trace directly
 * back to the appropriate location in the model.  The basic format
 * is <system>/block_name, where system is the system number (uniquely
 * assigned by Simulink) and block_name is the name of the block.
 *
 * Use the MATLAB hilite_system command to trace the generated code back
 * to the model.  For example,
 *
 * hilite_system('<S3>')    - opens system 3
 * hilite_system('<S3>/Kp') - opens and selects block Kp which resides in S3
 *
 * Here is the system hierarchy for this model
 *
 * '<Root>' : 'pend_ctrl_lin'
 * '<S1>'   : 'pend_ctrl_lin/B&R reference input'
 * '<S2>'   : 'pend_ctrl_lin/Configurable Controller  Subsystem1'
 * '<S3>'   : 'pend_ctrl_lin/inverted_pendulum_IOs'
 * '<S4>'   : 'pend_ctrl_lin/Configurable Controller  Subsystem1/State Feedback Controller (blks)'
 */
#endif                                 /* RTW_HEADER_pend_ctrl_lin_h_ */
```

#### pend_ctrl_lin_private.h
```c
/********************************************************************
 * COPYRIGHT -- Bernecker + Rainer Industrie-Elektronik Ges.m.b.H.
 ********************************************************************
 * Program: pend_ctrl_lin
 * File: pend_ctrl_lin_private.h
 * Author: Bernecker + Rainer Industrie Elektronik Ges.m.b.H.
 * Created: Wed Mar 17 14:21:47 2010
 ********************************************************************
 * Header for program pend_ctrl_lin
 ********************************************************************
 * Generated with B&R Automation Studio Target for Simulink  V6.1.0
 * (ERT based)
 ********************************************************************/

#ifndef RTW_HEADER_pend_ctrl_lin_private_h_
#define RTW_HEADER_pend_ctrl_lin_private_h_
#include "rtwtypes.h"
#define _ASMATH_
#define ASMATH_
#define _ASMATH_H
#define ASMATH_H
#define _ASMATH_H_
#define ASMATH_H_
#define _ASSTRING_
#define ASSTRING_
#define _ASSTRING_H
#define ASSTRING_H
#define _ASSTRING_H_
#define ASSTRING_H_
#include <bur/plctypes.h>
#ifdef _DEFAULT_INCLUDES
#include <AsDefault.h>
#endif

#ifndef MIN
#define MIN(a,b)                       ((a) < (b) ? (a) : (b))
#endif

#ifndef MAX
#define MAX(a,b)                       ((a) > (b) ? (a) : (b))
#endif
#endif                                 /* RTW_HEADER_pend_ctrl_lin_private_h_ */
```

#### pend_ctrl_lin_types.h
```c
/********************************************************************
 * COPYRIGHT -- Bernecker + Rainer Industrie-Elektronik Ges.m.b.H.
 ********************************************************************
 * Program: pend_ctrl_lin
 * File: pend_ctrl_lin_types.h
 * Author: Bernecker + Rainer Industrie Elektronik Ges.m.b.H.
 * Created: Wed Mar 17 14:21:47 2010
 ********************************************************************
 * Header for program pend_ctrl_lin
 ********************************************************************
 * Generated with B&R Automation Studio Target for Simulink  V6.1.0
 * (ERT based)
 ********************************************************************/

#ifndef RTW_HEADER_pend_ctrl_lin_types_h_
#define RTW_HEADER_pend_ctrl_lin_types_h_
#ifndef MIN
#define MIN(a,b)                       ((a) < (b) ? (a) : (b))
#endif

#ifndef MAX
#define MAX(a,b)                       ((a) > (b) ? (a) : (b))
#endif

/* Forward declaration for rtModel */
typedef struct tag_RTM_pend_ctrl_lin RT_MODEL_pend_ctrl_lin;

#endif                                 /* RTW_HEADER_pend_ctrl_lin_types_h_ */
```

#### rtwtypes.h
```c
/********************************************************************
 * COPYRIGHT -- Bernecker + Rainer Industrie-Elektronik Ges.m.b.H.
 ********************************************************************
 * Program: pend_ctrl_lin
 * File: rtwtypes.h
 * Author: Bernecker + Rainer Industrie Elektronik Ges.m.b.H.
 * Created: Wed Mar 17 14:21:47 2010
 ********************************************************************
 * Header for program pend_ctrl_lin
 ********************************************************************
 * Generated with B&R Automation Studio Target for Simulink  V6.1.0
 * (ERT based)
 ********************************************************************/

#ifndef RTWTYPES_H
#define RTWTYPES_H

/* Logical type definitions */
#if (!defined(__cplusplus))
#  ifndef false
#   define false                       (0U)
#  endif

#  ifndef true
#   define true                        (1U)
#  endif
#endif

/*=======================================================================*
 * Target hardware information
 *   Device type: Intel->x86/Pentium
 *   Number of bits:     char:   8    short:   16    long:  32
 *                       long:  32
 *                       native word size:  32
 *   Byte ordering: LittleEndian
 *   Signed integer division rounds to: Zero
 *   Shift right on a signed integer as arithmetic shift: on
 *=======================================================================*/

/*=======================================================================*
 * Fixed width word size data types:                                     *
 *   int8_T, int16_T, int32_T     - signed 8, 16, or 32 bit integers     *
 *   uint8_T, uint16_T, uint32_T  - unsigned 8, 16, or 32 bit integers   *
 *   real32_T, real64_T           - 32 and 64 bit floating point numbers *
 *=======================================================================*/
typedef signed char int8_T;
typedef unsigned char uint8_T;
typedef short int16_T;
typedef unsigned short uint16_T;
typedef long int32_T;
typedef unsigned long uint32_T;
typedef float real32_T;
typedef double real64_T;

/*===========================================================================*
 * Generic type definitions: boolean_T, char_T, byte_T, int_T, uint_T,       *
 *                           real_T, time_T, ulong_T.                        *
 *===========================================================================*/
typedef double real_T;
typedef double time_T;
typedef unsigned char boolean_T;
typedef long int_T;
typedef unsigned long uint_T;
typedef unsigned long ulong_T;
typedef char char_T;
typedef unsigned char uchar_T;
typedef char_T byte_T;

/*=======================================================================*
 * Min and Max:                                                          *
 *   int8_T, int16_T, int32_T     - signed 8, 16, or 32 bit integers     *
 *   uint8_T, uint16_T, uint32_T  - unsigned 8, 16, or 32 bit integers   *
 *=======================================================================*/
#define MAX_int8_T                     ((int8_T)(127))
#define MIN_int8_T                     ((int8_T)(-128))
#define MAX_uint8_T                    ((uint8_T)(255U))
#define MAX_int16_T                    ((int16_T)(32767))
#define MIN_int16_T                    ((int16_T)(-32768))
#define MAX_uint16_T                   ((uint16_T)(65535U))
#define MAX_int32_T                    ((int32_T)(2147483647))
#define MIN_int32_T                    ((int32_T)(-2147483647-1))
#define MAX_uint32_T                   ((uint32_T)(0xFFFFFFFFU))

/* Block D-Work pointer type */
typedef void * pointer_T;

#endif                                 /* RTWTYPES_H */

#ifndef MIN
#define MIN(a,b)                       ((a) < (b) ? (a) : (b))
#endif

#ifndef MAX
#define MAX(a,b)                       ((a) > (b) ? (a) : (b))
#endif
```

#### task_properties.txt
```
For manual assignment to hardware configuration please
add the following additional include directories:

\Logical\MATLAB_includes\R2019b\

And the following additional build options:

-lm -D MODEL=pend_ctrl_lin -D NUMST=1 -D NCSTATES=0 -D HAVESTDIO -D MODEL_HAS_DYNAMICALLY_LOADED_SFCNS=0 -D CLASSIC_INTERFACE=0 -D ALLOCATIONFCN=0 -D TID01EQ=0 -D TERMFCN=1 -D ONESTEPFCN=0 -D MAT_FILE=0 -D MULTI_INSTANCE_CODE=0 -D INTEGER_CODE=0 -D MT=0
```

#### multiword_types.h - not listed in the package file held
```c
/********************************************************************
 * COPYRIGHT -- Bernecker + Rainer Industrie-Elektronik Ges.m.b.H.
 ********************************************************************
 * Program: pend_ctrl_lin
 * File: multiword_types.h
 * Author: Bernecker + Rainer Industrie Elektronik Ges.m.b.H.
 * Created: Wed Mar 17 14:21:47 2010
 ********************************************************************
 * Header for program pend_ctrl_lin
 ********************************************************************
 * Generated with B&R Automation Studio Target for Simulink  V6.1.0
 * (ERT based)
 ********************************************************************/

#ifndef MULTIWORD_TYPES_H
#define MULTIWORD_TYPES_H
#include "rtwtypes.h"

/*
 * Definitions supporting external data access
 */
typedef int32_T chunk_T;
typedef uint32_T uchunk_T;

#endif                                 /* MULTIWORD_TYPES_H */

#ifndef MIN
#define MIN(a,b)                       ((a) < (b) ? (a) : (b))
#endif

#ifndef MAX
#define MAX(a,b)                       ((a) > (b) ? (a) : (b))
#endif
```

#### pend_ctrl_lin_dt.h - not listed in the package file held
```c
/*
 * pend_ctrl_lin_dt.h
 *
 * Academic License - for use in teaching, academic research, and meeting
 * course requirements at degree granting institutions only.  Not for
 * government, commercial, or other organizational use.
 *
 * Code generation for model "pend_ctrl_lin".
 *
 * Model version              : 1.180
 * Simulink Coder version : 9.2 (R2019b) 18-Jul-2019
 * C source code generated on : Fri Apr  1 12:06:09 2022
 *
 * Target selection: bur_ert.tlc
 * Embedded hardware selection: Intel->x86/Pentium
 * Code generation objectives: Unspecified
 * Validation result: Not run
 */

#include "ext_types.h"

/* data type size table */
static uint_T rtDataTypeSizes[] = {
  sizeof(real_T),
  sizeof(real32_T),
  sizeof(int8_T),
  sizeof(uint8_T),
  sizeof(int16_T),
  sizeof(uint16_T),
  sizeof(int32_T),
  sizeof(uint32_T),
  sizeof(boolean_T),
  sizeof(fcn_call_T),
  sizeof(int_T),
  sizeof(pointer_T),
  sizeof(action_T),
  2*sizeof(uint32_T)
};

/* data type name table */
static const char_T * rtDataTypeNames[] = {
  "real_T",
  "real32_T",
  "int8_T",
  "uint8_T",
  "int16_T",
  "uint16_T",
  "int32_T",
  "uint32_T",
  "boolean_T",
  "fcn_call_T",
  "int_T",
  "pointer_T",
  "action_T",
  "timer_uint32_pair_T"
};

/* data type transitions for block I/O structure */
static DataTypeTransition rtBTransitions[] = {
  { (char_T *)(&pend_ctrl_lin_B.Input1[0]), 0, 0, 10 }
  ,

  { (char_T *)(&pend_ctrl_lin_DWork.Outputxtheta_PWORK.LoggedData), 11, 0, 4 }
};

/* data type transition table for block I/O structure */
static DataTypeTransitionTable rtBTransTable = {
  2U,
  rtBTransitions
};

/* [EOF] pend_ctrl_lin_dt.h */
```

#### bur_logging.c
```c
/********************************************************************
 * COPYRIGHT -- Bernecker + Rainer
 ********************************************************************
 * File: bur_logging.c
 * Author: B&R
 * Created: September 07, 2010
 * Abstract: This is a simple logger module to log data by using
 * the library 'AsArLog'. The needed FBK's work asynchronously so
 * buffering the entries is necessary. The buffer 'entry_buffer'
 * is realized as FIFO- buffer (circular- buffer) an is able to
 * contain 'NUM_LOG_ENTRIES' entries at once (per default 5),
 * each combined with a ASCII- string of 'LOG_STRSIZE' length
 * (per default 128, including the logging- header (modelname plus
 * a few other char's) and trailing zero- byte).
 *******************************************************************/

#include "bur_logging.h"
#include <AsArLog.h>
#include <string.h>

/** defines **/

/*  Ident for the AR logger module to be written.
    The default logger module is base user module "$arlogusr". */
#ifndef LOG_IDENT
# define LOG_IDENT (arlogBASE_USER_LOG_IDENT)
#endif

/* size of the entry- buffer */
#ifndef NUM_LOG_ENTRIES
# define NUM_LOG_ENTRIES (5U)
#endif

/* length of ascii- string per log- entry */
#ifndef LOG_STRSIZE
# define LOG_STRSIZE (128U)
#endif

#ifndef MODEL
# define MODEL no_modelname_specified
#endif

/* Get Modelname as string (used for the logging- header) */
#define MODEL_STRING GET_STRING(MODEL)

/* needed to expand the modelname */
#define GET_STRING(arg) GET_STRING1(arg)
#define GET_STRING1(arg) #arg

/** typedefs **/

/* Container for one log- etnry */
typedef struct
{
    logLevel_t  logLevel;
    UDINT       errornr;
    char        asciiString[LOG_STRSIZE];
}logEntry_t;

/** local data **/

static AsArLogWrite_typ 	logWrite_var;

/*  Entry- buffer to temporary store entries before written
    to a logger module */
static logEntry_t entry_buffer[NUM_LOG_ENTRIES];

/*  buffer_first marks the position of the next entry to be
    written to a logger module. (The 'begin' or 'start' of
    the circular- buffer)

    buffer_load is the number of entries currently stored in
    the entry buffer */
static size_t buffer_first = 0, buffer_load = 0;

/** end local data **/

/** local function prototypes **/

static void init_writeFirst();
static void createLogHeader(char *string);

/** end local function prototypes **/

/** public functions **/

BOOL writeLogEntry( logLevel_t logLevel,
                    UDINT errornr,
                    const char* string)
{
    if(buffer_load < NUM_LOG_ENTRIES)
    { /* There's still some space available in the buffer,
         so write the logging information */

        /*  Remaining chars exkluding the trailing zero- byte */
        size_t charsRemaining;

        /* Index to store data into (next free position) */
        size_t tmpIndex = (buffer_first+buffer_load)%NUM_LOG_ENTRIES;
        logEntry_t *tmpEntry = &entry_buffer[tmpIndex];

        /* copy logLevel to the buffer */
        switch(logLevel)
        {
            case logLevel_info:
                tmpEntry->logLevel = arlogLEVEL_INFO;
                break;

            case logLevel_warning:
                tmpEntry->logLevel = arlogLEVEL_WARNING;
                break;

            case logLevel_fatal:
                tmpEntry->logLevel = arlogLEVEL_FATAL;
                break;

            default:
                tmpEntry->logLevel = arlogLEVEL_INFO;
                break;
        }

        /* copy errornr to the buffer */
        tmpEntry->errornr  = errornr;

        /* Create the log- header:  "Model 'Modelname': "   */
        createLogHeader(tmpEntry->asciiString);

        charsRemaining = LOG_STRSIZE - (strlen(tmpEntry->asciiString)+1);

        /* copy string (if present) to the buffer */
        if( (string != NULL) && (charsRemaining > 0) )
        {
            /* copy the error- string to the buffer */
            strncat(tmpEntry->asciiString, string, charsRemaining);
        }

        /* assure that the string is at least null- terminated */
        tmpEntry->asciiString[LOG_STRSIZE-1] = '\0';

        buffer_load++;
        return TRUE;
    }
    /* 'else' the buffer is full, so return FALSE */
    return FALSE;
}

UINT loggingWork()
{
    static BOOL logInProgress = FALSE;
    long count=0;

    for(count=0; count<2; count++)
    {
        if(logInProgress)
        {   /*  logging is currently in progress
                --> call the FBK */
            AsArLogWrite(&logWrite_var);
            if(logWrite_var.status == ERR_OK); /* do nothing */
            else if(logWrite_var.status == ERR_FUB_BUSY)
            {
                /*  FBK is busy --> retry next time */
                return ERR_FUB_BUSY;

            }
            else
            {
                /* an error occurred somewhere */
                return logWrite_var.status;
            }

            /* ERR_OK */
            buffer_load--;
            buffer_first = (buffer_first+1) % NUM_LOG_ENTRIES;
            logInProgress = FALSE;
        }

        /* no logging in progress --> check if there's another entry in the buffer */
        if(buffer_load > 0)
        {
            init_writeFirst();
            logInProgress = TRUE;
        }

    } /* end for(...) */

    return (logInProgress ? ERR_FUB_BUSY : ERR_OK);

} /* end loggingWork() */

/** end public functions **/

/** local functions **/

/*  Initialize the instance- variable of the AsArLogWrite(...) FBK
    with the next entry from the entry- buffer */
static void init_writeFirst()
{
	logWrite_var.enable 	= TRUE;
	logWrite_var.ident		= LOG_IDENT;
	logWrite_var.logLevel	= entry_buffer[buffer_first].logLevel;
	logWrite_var.errornr	= entry_buffer[buffer_first].errornr;
	logWrite_var.mem		= (UDINT)NULL;
	logWrite_var.len		= 0;
	logWrite_var.asciiString= (UDINT)entry_buffer[buffer_first].asciiString;
}

static void createLogHeader(char *string)
{
/*  Remaining chars exkluding the trailing zero- byte */
    size_t charsRemaining;

    if(string == NULL)return;

    /* mark as empty string */
    string[0] = '\0';
    strcat(string, "Model \'");

    /*  remaining chars. The '1' in (strlen(string)+1)
        is for the trailing zero- byte */
    charsRemaining = LOG_STRSIZE - (strlen(string)+1);
    if(charsRemaining > 0)
        strncat(string, MODEL_STRING, charsRemaining);

    charsRemaining = LOG_STRSIZE - (strlen(string)+1);
    if(charsRemaining > 0)
        strncat(string, "\': ", charsRemaining);
}

/** end local functions **/
```

#### bur_logging.h
```c
/********************************************************************
 * COPYRIGHT -- Bernecker + Rainer
 ********************************************************************
 * File: bur_logging.h
 * Author: B&R
 * Created: September 07, 2010
 *******************************************************************/

#include <bur/plctypes.h>
#ifdef _DEFAULT_INCLUDES
 #include <AsDefault.h>
#endif

#ifndef TRUE
# define TRUE  (1U)
#endif

#ifndef FALSE
# define FALSE (0U)
#endif

/** public datatypes **/

/*  The three different types of log- entries
    according to the three types of log- entries
    in 'AsArLog'. */
typedef enum
{
	logLevel_info,
	logLevel_warning,
	logLevel_fatal
}logLevel_t;

/** end public datatypes **/

/** public function prototypes **/

/* call this function to add a new logging- entry */
BOOL writeLogEntry( logLevel_t logLevel,
                    UDINT errornr,
                    const char* string);

/* poll this function to write the entries to the log-files */
UINT loggingWork();

/** end public function prototypes **/
```
